INTERFACE iDM_DriveHealth

METHOD Disable : BOOL
VAR_INPUT
END_VAR
END_METHOD

METHOD Enable : BOOL
VAR_INPUT
END_VAR
END_METHOD

PROPERTY FaultLocation : STRING(50)
GET
END_GET
END_PROPERTY

PROPERTY HasFault : BOOL
GET
END_GET
END_PROPERTY

PROPERTY IsReady : BOOL
GET
END_GET
END_PROPERTY

PROPERTY IsRunning : BOOL
GET
END_GET
END_PROPERTY

METHOD Reset : BOOL
VAR_INPUT
END_VAR
END_METHOD

END_INTERFACE

(* stored: Version 1.1.0.1, ProductVersion 3.1.4024.16
   Itf iDM_DriveHealth: Id {fcb5f53a-de9a-4459-8915-1d4c6680bd48}
   Method Disable: Id {0a7cca81-e8cf-4a5f-bde0-ccd9352d9e9c}
   Method Enable: Id {1b8f1800-5961-4994-a5dc-4bd60308b993}
   Property FaultLocation: Id {bd616e79-31c8-4788-8227-3a8af4566b61}
   Get Get: Id {841784e1-86f2-41f3-a77d-83e598e2c01c}
   Property HasFault: Id {0d4baedf-1bc0-4914-8cdf-7f8c7cd7f777}
   Get Get: Id {cadfc129-9100-42d1-8b40-e61b84bd35af}
   Property IsReady: Id {486b553b-168e-4191-88a6-86601dd17b47}
   Get Get: Id {4fefba3a-51f9-4e3b-a03e-224f986d0e9e}
   Property IsRunning: Id {2e7d3f9f-a409-4733-85cd-9d9dfcb594a3}
   Get Get: Id {b145d479-34fa-45b2-aee1-144c7c6c12bd}
   Method Reset: Id {9f0533d5-aa48-4501-99fb-f112d3854da0} *)
